TEXTLIST TextList_TrackState
  0 = 'Ready'
  10 = 'スタート地点へ移動指令'
  11 = 'スタート位置移動確認'
  20 = '充填位置へ移動指令'
  21 = '充填位置移動'
  30 = 'キャップ位置へ移動指令'
  31 = 'キャップ位置移動'
  32 = 'キャップ締め回転指令'
  33 = 'キャップ締め回転'
  40 = '待機場所へ移動指令'
  41 = '待機場所へ移動'
   = ''
END_TEXTLIST

(* stored: Version 1.1.0.1
   TextList TextList_TrackState: Id {e8576e3c-81f2-4ea5-bb26-857fff8f2c4c} *)
